# B&R Automation Studio project NAEUL004C00R13L518F00 (part 50)

#### Act_Main.st - Do Not Change!!!
```iecst
(** 2020-05-26 **)
ACTION Act_Main:

	//Main
IF bModuleNotOK = FALSE THEN

		CASE eStat OF

			AWActIdle:
				IF eStatus <> Idle THEN	//Reset Data
					//Private
					fbStop(bEn := FALSE);
					fbRstAxisErr(bEn := FALSE);
					fbJog(bEn := FALSE);
					fbMovRel(bEn := FALSE);
					fbMovAbs(bEn := FALSE);
					fbHoming(bEn := FALSE);
					fbPwrOff(bEn := FALSE);
					fbPwrOn(bEn := FALSE);
					fbFullHm(bEn := FALSE);
					fbFullMovAbs(bEn := FALSE);
					fbFullMovAbsBl(bEn := FALSE);
					fbSDOWrite(bEn := FALSE);
					fbTm(IN := FALSE);
					usiStep				:= 0;
					usiCount			:= 0;
					bNotInterruptible	:= FALSE;
					tyParamOutDriver.uiCtrlword_6040.7	:= FALSE;
					sStatTxt	:= a_sStatText[eStat];

				END_IF

				eStatus	:= Idle;

				IF EDGENEG(p_bManual) THEN
					fMotionCANRstCtrlWord(ADR(tyParamOutDriver));
				END_IF

			AWActGoWidth:
				IF (eStatus = Idle OR eStatus = Busy) THEN

					eStatus	:= Busy;

					sStatTxt	:= a_sStatText[eStat];

					bNotInterruptible	:= TRUE;

					CASE usiStep OF
						0:	//Wait For Motion Parameter Update
							p_diMovePosInUM	:= ABS(fAWWidthToPosInUM(p_diGoWidth , p_diWidthAtHmPos));
							usiStep	:= 1;

						1:	//Check Position Difference
							IF tyParamOut.bPosDiff = TRUE THEN
								usiStep	:= 2;
							ELSE
								eStatus	:= Done;
							END_IF

						2:	//Move
							fbFullMovAbsBl.tyParamInDriver					:= tyParamInDriver;
							fbFullMovAbsBl.tyParamInMove.diPosInUM			:= p_diMovePosInUM;
							fbFullMovAbsBl.tyParamInMove.diDistInUM			:= p_diMoveDistInUM;
							fbFullMovAbsBl.tyParamInMove.diVelInUMPS		:= p_diMoveVelInUMPS;
							fbFullMovAbsBl.tyParamInMove.diAcc				:= p_diMoveAcc;
							fbFullMovAbsBl.tyParamInMove.diDec				:= p_diMoveDec;
							fbFullMovAbsBl.tyParamOut						:= tyParamOut;
							fbFullMovAbsBl(bEn := TRUE);

							IF fbFullMovAbsBl.udiStatus = 0 THEN
								eStatus	:= Done;
							ELSIF fbFullMovAbsBl.udiStatus < 65534 THEN
								eStatus		:= Error;

								IF fbFullMovAbsBl.udiStatus = 1401 THEN
									udiStatus	:= 10002;	//Power On Time Out While Going New Width
								ELSIF fbFullMovAbsBl.udiStatus = 1402 THEN
									udiStatus	:= 10003;	//Homing Time Out While Going New Width
								ELSIF fbFullMovAbsBl.udiStatus = 1403 THEN
									udiStatus	:= 10004;	//Move Absolute Time Out While Going New Width
								ELSIF fbFullMovAbsBl.udiStatus = 1405 THEN
									udiStatus	:= 10005;	//Stop Motion Time Out While Going New Width
								ELSIF fbFullMovAbsBl.udiStatus = 1408 THEN
									udiStatus	:= 10006;	//Axis Error Reset Failed While Going New Width
								ELSIF fbFullMovAbsBl.udiStatus = 1409 THEN
									udiStatus	:= 10007;	//Axis Error Occur In Move Absolute While Going New Width
								ELSIF fbFullMovAbsBl.udiStatus = 1411 THEN
									udiStatus	:= 10008;	//Axis Error Occur In Homing While Going New Width
								ELSIF fbFullMovAbsBl.udiStatus = 1412 THEN
									udiStatus	:= 10009;	//Homing Done But Home Flag Is Not Activated While Going New Width
								ELSIF fbFullMovAbsBl.udiStatus = 1413 THEN
									udiStatus	:= 10010;	//Forward Limit Activated In Homing While Going New Width
								ELSIF fbFullMovAbsBl.udiStatus = 1414 THEN
									udiStatus	:= 10011;	//Reverse Limit Activated In Homing While Going New Width
								ELSIF fbFullMovAbsBl.udiStatus = 1415 THEN
									udiStatus	:= 10012;	//Forward Limit Activated In Move Absolute While Going New Width
								ELSIF fbFullMovAbsBl.udiStatus = 1416 THEN
									udiStatus	:= 10013;	//Reverse Limit Activated In Move Absolute While Going New Width
								ELSE
									udiStatus	:= fbFullMovAbsBl.udiStatus;
								END_IF
							END_IF

					END_CASE

				END_IF

			AWActGoWidthOff:
				IF (eStatus = Idle OR eStatus = Busy) THEN

					eStatus	:= Busy;

					sStatTxt	:= a_sStatText[eStat];

					bNotInterruptible	:= TRUE;

					CASE usiStep OF
						0:	//Wait For Motion Parameter Update
							p_diMovePosInUM	:= ABS(fAWWidthToPosInUM(p_diGoWidth , p_diWidthAtHmPos));
							usiStep	:= 1;

						1:	//Check Position Difference
							IF tyParamOut.bPosDiff = TRUE THEN
								usiStep	:= 2;
							ELSE
								eStatus	:= Done;
							END_IF

						2:	//Move
							fbFullMovAbsBl.tyParamInDriver					:= tyParamInDriver;
							fbFullMovAbsBl.tyParamInMove.diPosInUM			:= p_diMovePosInUM;
							fbFullMovAbsBl.tyParamInMove.diDistInUM			:= p_diMoveDistInUM;
							fbFullMovAbsBl.tyParamInMove.diVelInUMPS		:= p_diMoveVelInUMPS;
							fbFullMovAbsBl.tyParamInMove.diAcc				:= p_diMoveAcc;
							fbFullMovAbsBl.tyParamInMove.diDec				:= p_diMoveDec;
							fbFullMovAbsBl.tyParamOut						:= tyParamOut;
							fbFullMovAbsBl(bEn := TRUE);

							IF fbFullMovAbsBl.udiStatus = 0 THEN
								usiStep	:= 3;
							ELSIF fbFullMovAbsBl.udiStatus < 65534 THEN
								eStatus		:= Error;

								IF fbFullMovAbsBl.udiStatus = 1401 THEN
									udiStatus	:= 10035;	//Power On Time Out While Going New Width And Off
								ELSIF fbFullMovAbsBl.udiStatus = 1402 THEN
									udiStatus	:= 10036;	//Homing Time Out While Going New Width And Off
								ELSIF fbFullMovAbsBl.udiStatus = 1403 THEN
									udiStatus	:= 10037;	//Move Absolute Time Out While Going New Width And Off
								ELSIF fbFullMovAbsBl.udiStatus = 1405 THEN
									udiStatus	:= 10038;	//Stop Motion Time Out While Going New Width And Off
								ELSIF fbFullMovAbsBl.udiStatus = 1408 THEN
									udiStatus	:= 10039;	//Axis Error Reset Failed While Going New Width And Off
								ELSIF fbFullMovAbsBl.udiStatus = 1409 THEN
									udiStatus	:= 10040;	//Axis Error Occur In Move Absolute While Going New Width And Off
								ELSIF fbFullMovAbsBl.udiStatus = 1411 THEN
									udiStatus	:= 10041;	//Axis Error Occur In Homing While Going New Width And Off
								ELSIF fbFullMovAbsBl.udiStatus = 1412 THEN
									udiStatus	:= 10042;	//Homing Done But Home Flag Is Not Activated While Going New Width And Off
								ELSIF fbFullMovAbsBl.udiStatus = 1413 THEN
									udiStatus	:= 10043;	//Forward Limit Activated In Homing While Going New Width And Off
								ELSIF fbFullMovAbsBl.udiStatus = 1414 THEN
									udiStatus	:= 10044;	//Reverse Limit Activated In Homing While Going New Width And Off
								ELSIF fbFullMovAbsBl.udiStatus = 1415 THEN
									udiStatus	:= 10045;	//Forward Limit Activated In Move Absolute While Going New Width And Off
								ELSIF fbFullMovAbsBl.udiStatus = 1416 THEN
									udiStatus	:= 10046;	//Reverse Limit Activated In Move Absolute While Going New Width And Off
								ELSE
									udiStatus	:= fbFullMovAbsBl.udiStatus;
								END_IF
							END_IF

						3:	//Turn Off Motor
							fMotionCANRstCtrlWord(ADR(tyParamOutDriver));
							eStatus	:= Done;

					END_CASE

				END_IF

			AWActFullHm:
				IF (eStatus = Idle OR eStatus = Busy) THEN

					eStatus	:= Busy;

					sStatTxt	:= a_sStatText[eStat];

					bNotInterruptible	:= TRUE;

					fbFullHm.tyParamInDriver	:= tyParamInDriver;
					fbFullHm.tyParamOut			:= tyParamOut;
					fbFullHm(bEn := TRUE);

					IF fbFullHm.udiStatus = 0 THEN
						eStatus	:= Done;
					ELSIF fbFullHm.udiStatus < 65534 THEN
						eStatus		:= Error;

						IF fbFullHm.udiStatus = 1401 THEN
							udiStatus	:= 10014;	//Power On Time Out While Full Homing
						ELSIF fbFullHm.udiStatus = 1402 THEN
							udiStatus	:= 10015;	//Homing Time Out While Full Homing
						ELSIF fbFullHm.udiStatus = 1405 THEN
							udiStatus	:= 10016;	//Stop Motion Time Out While Full Homing
						ELSIF fbFullHm.udiStatus = 1408 THEN
							udiStatus	:= 10017;	//Axis Error Reset Failed While Full Homing
						ELSIF fbFullHm.udiStatus = 1411 THEN
							udiStatus	:= 10018;	//Axis Error Occur In Homing While Full Homing
						ELSIF fbFullHm.udiStatus = 1412 THEN
							udiStatus	:= 10019;	//Homing Done But Home Flag Is Not Activated While Full Homing
						ELSIF fbFullHm.udiStatus = 1413 THEN
							udiStatus	:= 10020;	//Forward Limit Activated In Homing While Full Homing
						ELSIF fbFullHm.udiStatus = 1414 THEN
							udiStatus	:= 10021;	//Reverse Limit Activated In Homing While Full Homing
						ELSE
							udiStatus	:= fbFullHm.udiStatus;
						END_IF
					END_IF

				END_IF

			AWActPwrOn:
				IF (eStatus = Idle OR eStatus = Busy) THEN

					eStatus	:= Busy;

					sStatTxt	:= a_sStatText[eStat];

					fbPwrOn.tyParamInDriver	:= tyParamInDriver;
					fbPwrOn(bEn := TRUE);

					IF fbPwrOn.udiStatus = 0 THEN
						eStatus	:= Done;
					ELSIF fbPwrOn.udiStatus < 65534 THEN
						eStatus		:= Error;

						IF fbPwrOn.udiStatus = 1401 THEN
							udiStatus	:= 10022;	//Power On Time Out
						ELSE
							udiStatus	:= fbPwrOn.udiStatus;
						END_IF
					END_IF

				END_IF

			AWActPwrOff:
				IF (eStatus = Idle OR eStatus = Busy) THEN

					eStatus	:= Busy;

					sStatTxt	:= a_sStatText[eStat];

					fbPwrOff.tyParamInDriver	:= tyParamInDriver;
					fbPwrOff(bEn := TRUE);

					IF fbPwrOff.udiStatus = 0 THEN
						eStatus	:= Done;
					ELSIF fbPwrOff.udiStatus < 65534 THEN
						eStatus		:= Error;

						IF fbPwrOff.udiStatus = 1400 THEN
							udiStatus	:= 10023;	//Power Off Time Out
						ELSE
							udiStatus	:= fbPwrOff.udiStatus;
						END_IF
					END_IF

				END_IF

			AWActHoming:

				IF (eStatus = Idle OR eStatus = Busy) THEN

					eStatus	:= Busy;

					sStatTxt	:= a_sStatText[eStat];

					bNotInterruptible	:= TRUE;

					fbHoming.tyParamInDriver	:= tyParamInDriver;
					fbHoming.tyParamOut			:= tyParamOut;
					fbHoming(bEn := TRUE);

					IF fbHoming.udiStatus = 0 THEN
						eStatus	:= Done;
					ELSIF fbHoming.udiStatus < 65534 THEN
						eStatus		:= Error;

						IF fbHoming.udiStatus = 1402 THEN
							udiStatus	:= 10024;	//Homing Time Out
						ELSIF fbHoming.udiStatus = 1411 THEN
							udiStatus	:= 10018;	//Axis Error Occur In Homing While Full Homing

						ELSIF fbHoming.udiStatus = 1413 THEN
							udiStatus	:= 10020;	//Forward Limit Activated In Homing While Full Homing
						ELSIF fbHoming.udiStatus = 1414 THEN
							udiStatus	:= 10021;	//Reverse Limit Activated In Homing While Full Homing
						ELSE
							udiStatus	:= fbHoming.udiStatus;
						END_IF
					END_IF

				END_IF

			AWActMovAbs:
				IF (eStatus = Idle OR eStatus = Busy) THEN

					eStatus	:= Busy;

					sStatTxt	:= a_sStatText[eStat];

					bNotInterruptible	:= TRUE;

					fbMovAbs.tyParamInDriver			:= tyParamInDriver;
					fbMovAbs.tyParamInMove.diPosInUM	:= p_diMovePosInUM;
					fbMovAbs.tyParamInMove.diDistInUM	:= p_diMoveDistInUM;
					fbMovAbs.tyParamInMove.diVelInUMPS	:= p_diMoveVelInUMPS;
					fbMovAbs.tyParamInMove.diAcc		:= p_diMoveAcc;
					fbMovAbs.tyParamInMove.diDec		:= p_diMoveDec;
					fbMovAbs(bEn := TRUE);

					IF fbMovAbs.udiStatus = 0 THEN
						eStatus	:= Done;
					ELSIF fbMovAbs.udiStatus < 65534 THEN
						eStatus		:= Error;

						IF fbMovAbs.udiStatus = 1403 THEN
							udiStatus	:= 10025;	//Move Absolute Time Out
						ELSE
							udiStatus	:= fbMovAbs.udiStatus;
						END_IF
					END_IF

				END_IF

			AWActMovRel:
				IF (eStatus = Idle OR eStatus = Busy) THEN

					eStatus	:= Busy;

					sStatTxt	:= a_sStatText[eStat];

					bNotInterruptible	:= TRUE;

					fbMovRel.tyParamInDriver			:= tyParamInDriver;
					fbMovRel.tyParamInMove.diPosInUM	:= p_diMovePosInUM;
					fbMovRel.tyParamInMove.diDistInUM	:= p_diMoveDistInUM;
					fbMovRel.tyParamInMove.diVelInUMPS	:= p_diMoveVelInUMPS;
					fbMovRel.tyParamInMove.diAcc		:= p_diMoveAcc;
					fbMovRel.tyParamInMove.diDec		:= p_diMoveDec;
					fbMovRel(bEn := TRUE);

					IF fbMovRel.udiStatus = 0 THEN
						eStatus	:= Done;
					ELSIF fbMovRel.udiStatus < 65534 THEN
						eStatus		:= Error;

						IF fbMovRel.udiStatus = 1404 THEN
							udiStatus	:= 10026;	//Move Relative Time Out
						ELSE
							udiStatus	:= fbMovRel.udiStatus;
						END_IF
					END_IF

				END_IF

			AWActJogOpen:
				IF (eStatus = Idle OR eStatus = Busy) THEN

					eStatus	:= Busy;

					sStatTxt	:= a_sStatText[eStat];

					bNotInterruptible	:= TRUE;

					fbJog.tyParamInDriver	:= tyParamInDriver;
					fbJog.tyParamInMove.diAcc		:= p_diMoveAcc;
					fbJog.tyParamInMove.diDec		:= p_diMoveDec;

					IF p_bDir = TRUE THEN
						fbJog.tyParamInJog.diVelInUMPS	:= p_diJogVelInUMPS * -1;
					ELSE
						fbJog.tyParamInJog.diVelInUMPS	:= p_diJogVelInUMPS;
					END_IF

					fbJog(bEn := TRUE);

					IF fbJog.udiStatus = 0 THEN
						bJogging	:= TRUE;
						bJogOpen	:= TRUE;
						eStatus		:= Done;
					ELSIF fbJog.udiStatus < 65534 THEN
						udiStatus	:= fbJog.udiStatus;
						eStatus		:= Error;
					END_IF

				END_IF

			AWActJogClose:
				IF (eStatus = Idle OR eStatus = Busy) THEN

					eStatus	:= Busy;

					sStatTxt	:= a_sStatText[eStat];

					bNotInterruptible	:= TRUE;

					fbJog.tyParamInDriver			:= tyParamInDriver;
					fbJog.tyParamInMove.diAcc		:= p_diMoveAcc;
					fbJog.tyParamInMove.diDec		:= p_diMoveDec;

					IF p_bDir = TRUE THEN
						fbJog.tyParamInJog.diVelInUMPS	:= p_diJogVelInUMPS;
					ELSE
						fbJog.tyParamInJog.diVelInUMPS	:= p_diJogVelInUMPS * -1;
					END_IF

					fbJog(bEn := TRUE);

					IF fbJog.udiStatus = 0 THEN
						bJogging	:= TRUE;
						bJogClose	:= TRUE;
						eStatus		:= Done;
					ELSIF fbJog.udiStatus < 65534 THEN
						udiStatus	:= fbJog.udiStatus;
						eStatus		:= Error;
					END_IF

				END_IF

			AWActJogStop:
				IF (eStatus = Idle OR eStatus = Busy) THEN

					sStatTxt	:= a_sStatText[eStat];

					fMotionCANJogStop(ADR(tyParamOutDriver));
					bJogging	:= FALSE;
					bJogClose	:= FALSE;
					bJogOpen	:= FALSE;
					eStatus	:= Done;

				END_IF

			AWActRstAxisErr:
				IF (eStatus = Idle OR eStatus = Busy) THEN

					eStatus	:= Busy;

					sStatTxt	:= a_sStatText[eStat];

					fbRstAxisErr(bEn := TRUE);

					IF fbRstAxisErr.udiStatus = 0 THEN
						eStatus	:= Done;
					ELSIF fbRstAxisErr.udiStatus < 65534 THEN
						udiStatus	:= fbRstAxisErr.udiStatus;
						eStatus		:= Error;
					END_IF

				END_IF

			AWActStop:
				IF (eStatus = Idle OR eStatus = Busy) THEN

					eStatus	:= Busy;

					sStatTxt	:= a_sStatText[eStat];

					fbStop.tyParamInDriver	:= tyParamInDriver;
					fbStop(bEn := TRUE);

					IF fbStop.udiStatus = 0 THEN
						bJogging	:= FALSE;
						bJogClose	:= FALSE;
						bJogOpen	:= FALSE;
						eStatus		:= Done;
					ELSIF fbStop.udiStatus < 65534 THEN
						eStatus		:= Error;

						IF fbStop.udiStatus = 1405 THEN
							udiStatus	:= 10027;	//Stop Motion Time Out
						ELSE
							udiStatus	:= fbStop.udiStatus;
						END_IF
					END_IF

				END_IF
		END_CASE
ELSE
	CASE eStat OF
		AWActSDOWrite:
			IF (eStatus = Idle OR eStatus = Busy) THEN

				eStatus	:= Busy;

				sStatTxt	:= a_sStatText[eStat];

				fbTm(IN := TRUE);

				IF fbTm.Q THEN

					fbSDOWrite.tyParamOut	:= tyParamOut;
					fbSDOWrite.tyTuning		:= p_tyTuning;

					fbSDOWrite(bEn := TRUE);

					IF fbSDOWrite.udiStatus = 0 THEN
						eStatus	:= Done;
					ELSIF fbSDOWrite.udiStatus < 65534 THEN
						fMotionCANRstCtrlWord(ADR(tyParamOutDriver));

						IF usiCount < 5 THEN
							fbTm(IN := FALSE);
							fbSDOWrite(bEn := FALSE);

							usiCount	:= usiCount + 1;
						ELSE
							eStatus	:= Error;

							IF fbSDOWrite.udiStatus = 1406 THEN
								udiStatus	:= 10028;	//SDO Write Error
							ELSE
								udiStatus	:= fbSDOWrite.udiStatus;
							END_IF
						END_IF

					END_IF

				END_IF

			END_IF

		AWActBGStartModOKChk:
			IF (eStatus = Idle OR eStatus = Busy) THEN

				sStatTxt	:= a_sStatText[eStat];

				bModuleOKChk	:= TRUE;
				eStatus			:= Done;

			END_IF

		AWActBGStopModOKChk:
			IF (eStatus = Idle OR eStatus = Busy) THEN

				sStatTxt	:= a_sStatText[eStat];

				bModuleOKChk	:= FALSE;
				eStatus			:= Done;

			END_IF

		AWActIdle:
			IF eStatus <> Idle THEN	//Reset Data
				//Private
				fbStop(bEn := FALSE);
				fbRstAxisErr(bEn := FALSE);
				fbJog(bEn := FALSE);
				fbMovRel(bEn := FALSE);
				fbMovAbs(bEn := FALSE);
				fbHoming(bEn := FALSE);
				fbPwrOff(bEn := FALSE);
				fbPwrOn(bEn := FALSE);
				fbFullHm(bEn := FALSE);
				fbFullMovAbs(bEn := FALSE);
				fbFullMovAbsBl(bEn := FALSE);
				fbSDOWrite(bEn := FALSE);
				fbTm(IN := FALSE);
				usiStep				:= 0;
				usiCount			:= 0;
				bNotInterruptible	:= FALSE;
				tyParamOutDriver.uiCtrlword_6040.7	:= FALSE;

				sStatTxt	:= a_sStatText[eStat];

			END_IF

			eStatus	:= Idle;

			IF EDGENEG(p_bManual) THEN
				fMotionCANRstCtrlWord(ADR(tyParamOutDriver));
			END_IF

		AWActRstNode:
			IF (eStatus = Idle OR eStatus = Busy) THEN

				eStatus	:= Busy;

				sStatTxt	:= a_sStatText[eStat];
				IF bRstErr THEN
					fbModuleOK(bEn := FALSE, bModuleOK := bModuleOK);
				END_IF
				fbModuleOK(bEn := TRUE);
				IF fbModuleOK.udiStatus = 0 THEN
					fbModuleOK(bEn := FALSE);
					eStatus			:= Done;
				ELSIF fbModuleOK.udiStatus < 65534 THEN
					eStatus		:= Error;

					IF fbModuleOK.udiStatus = 1407 THEN
						udiStatus	:= 10001;	//CANOpen Communication Error, ModuleOK Not TRUE
						fbModuleOK(bEn := FALSE);
					ELSE
						udiStatus	:= fbModuleOK.udiStatus;
					END_IF
				END_IF
			END_IF

		AWActRstAxisErr:
			IF (eStatus = Idle OR eStatus = Busy) THEN

				eStatus	:= Busy;

				sStatTxt	:= a_sStatText[eStat];

				fbRstAxisErr(bEn := TRUE);

				IF fbRstAxisErr.udiStatus = 0 THEN
					eStatus	:= Done;
				ELSIF fbRstAxisErr.udiStatus < 65534 THEN
					udiStatus	:= fbRstAxisErr.udiStatus;
					eStatus		:= Error;
				END_IF

			END_IF

	END_CASE
END_IF

END_ACTION
```

#### Act_Background.st - Do Not Change!!!
```iecst
(** 2020-05-26 **)
ACTION Act_Background:

	//Update Parameter
	IF bModuleOK = TRUE THEN

		tyParamInMove.diPosInUM		:= p_diMovePosInUM;
		tyParamInMove.diDistInUM	:= p_diMoveDistInUM;
		tyParamInMove.diVelInUMPS	:= p_diMoveVelInUMPS;
		tyParamInMove.diAcc			:= p_diMoveAcc;
		tyParamInMove.diDec			:= p_diMoveDec;

		fMotionCANUpdtDat(ADR(tyParamOut) , p_tyParamInConvert , tyParamOutDriver , tyParamInDriver , tyParamInMove , p_tyParamInHm , p_bDir, p_eNtParamMotorType);

		bWidthPosDiff	:= (tyParamOut.bIsHomed = FALSE) OR ((ABS((ABS(fAWWidthToPosInUM(p_diGoWidth , p_diWidthAtHmPos))) - tyParamOut.diActualPosInUM)) > 500);

		p_tyParamInConvert.diPitchInUM	:= fPitchCalc(p_diWidthOffsetInUM , p_diMaxWidthInUM , p_diMinWidthInUM , p_diPitchInUM);

		fbFullMovAbsBl.tyParamInConvert					:= p_tyParamInConvert;

		IF p_bDir = TRUE THEN
			bOpenSen	:= tyParamOut.bFwdLmtSen;
			bCloseSen	:= tyParamOut.bRevLmtSen;
		ELSE
			bOpenSen	:= tyParamOut.bRevLmtSen;
			bCloseSen	:= tyParamOut.bFwdLmtSen;
		END_IF

		CASE p_eNtParamMotorType OF
			DeltaAsdaA2:
				CASE tyParamOut.udiAxisErrID OF
					8976:	sAxisErrTxt	:= 'Over Current';
					12560:	sAxisErrTxt	:= 'Over Voltage';
					12576:	sAxisErrTxt	:= 'Under Voltage';
					12592:	sAxisErrTxt	:= 'Input Power Phase Loss';
					12816:	sAxisErrTxt	:= 'Regeneration Error';
					12848:	sAxisErrTxt	:= 'Overload';
					12849:	sAxisErrTxt	:= 'Pre-overload Warning';
					13056:	sAxisErrTxt	:= 'U,V,W Wiring Error';
					16912:	sAxisErrTxt	:= 'IGBT Temperature Error';
					21296:	sAxisErrTxt	:= 'Memory Error';
					21569:	sAxisErrTxt	:= 'Emergency Stop Activated';
					21570:	sAxisErrTxt	:= 'Forward Limit Switch Error';
					21571:	sAxisErrTxt	:= 'Reverse Limit Switch Error';
					21572:	sAxisErrTxt	:= 'Forward Software Limit';
					21573:	sAxisErrTxt	:= 'Reverse Software Limit';
					21760:	sAxisErrTxt	:= 'DSP Firmware Upgrade';
					25088:	sAxisErrTxt	:= 'CANopen SYNC Error';
					25360:	sAxisErrTxt	:= 'CANopen Data Initial Error';
					25376:	sAxisErrTxt	:= 'Adjustment Error';
					28961:	sAxisErrTxt	:= 'Motor Protection Error';
					28962:	sAxisErrTxt	:= 'Motor Error';
					29445:	sAxisErrTxt	:= 'Encoder Error';
					29446:	sAxisErrTxt	:= 'Encoder Output Error';
					29968:	sAxisErrTxt	:= 'Serial Communication Error';
					29984:	sAxisErrTxt	:= 'Serial Communication Time Out';
					33024:	sAxisErrTxt	:= 'CANbus Error (Bus-off)';
					33040:	sAxisErrTxt	:= 'CANopen SDO receive buffer overrun';
					33056:	sAxisErrTxt	:= 'CANbus Error (Warning)';
					33072:	sAxisErrTxt	:= 'Node Guarding or Heartbeat Error';
					33280:	sAxisErrTxt	:= 'CANopen PDO Object Error';
					33792:	sAxisErrTxt	:= 'Over Speed';
					34304:	sAxisErrTxt	:= 'Abnormal Pulse Control Command';
					34320:	sAxisErrTxt	:= 'Full Closed Loop Excessive Deviation';
					34321:	sAxisErrTxt	:= 'Excessive Deviation';
				END_CASE

			SchneiderLexium28:
				CASE tyParamOut.udiAxisErrID OF
					8724:	sAxisErrTxt	:= 'Over Current';
					8976:	sAxisErrTxt	:= 'Motor Overload';
					8977:	sAxisErrTxt	:= 'Drive overload (foldback)';
					9088:	sAxisErrTxt	:= 'Calculated offsets for current sensors out OF range';
					9089:	sAxisErrTxt := 'Motor phase missing';
					9090:	sAxisErrTxt := 'Overcurrent detected at one OF the digital outputs';
					12560:	sAxisErrTxt	:= 'DC Bus Over Voltage';
					12576:	sAxisErrTxt	:= 'DC Bus Under Voltage';
					12672:	sAxisErrTxt	:= 'Braking Resistor Overload';
					12673:	sAxisErrTxt	:= 'Safety function Safe Torque Off (STO) triggered';
					12674:	sAxisErrTxt	:= 'DC bus voltage measurement';
					12675:	sAxisErrTxt	:= 'Missing mains supply, undervoltage mains supply';
					12676:	sAxisErrTxt := 'The encoder supply voltage has dropped under operational value';
					12677:	sAxisErrTxt := 'The multi turn encoder battery voltage has dropped under 3 Vdc';
					12678:	sAxisErrTxt := 'Internal position synchronization error	detected between the multi turn AND the single turn modules';
					12679:	sAxisErrTxt := 'Generic error code of the multi turn module is detected';
					12697:	sAxisErrTxt := 'Braking resistor overload';
					16512:	sAxisErrTxt	:= 'Drive overtemperature (IPM)';
					16513:	sAxisErrTxt	:= 'Drive overtemperature (controller)';
					16534:	sAxisErrTxt := 'Temperature sensor inoperative';
					17168:	sAxisErrTxt	:= 'Power stage overtemperature';
					17280:	sAxisErrTxt := 'The encoder temperature is too high';
					17424:	sAxisErrTxt	:= 'Motor overtemperature';
					21808:	sAxisErrTxt	:= 'System error detected (nonvolatilememory)';
					21893:	sAxisErrTxt	:= 'Error detected in non-volatile memory';
					21889:	sAxisErrTxt	:= 'System error detected (nonvolatile memory)';
					21890:	sAxisErrTxt	:= 'System error detected (CAN power supply)';
					21891:	sAxisErrTxt	:= 'System error detected (selftest)';
					21894:	sAxisErrTxt	:= 'System error detected (NV ACCESS)';
					25472:	sAxisErrTxt	:= 'Target position rejected';
					25985:	sAxisErrTxt	:= 'System error detected(FPGA)';
					28816:	sAxisErrTxt	:= 'System error detected (FPGA does NOT match firmware)';
					28817:	sAxisErrTxt	:= 'Emergency Stop Activated';
					28961:	sAxisErrTxt := 'Motor blocked';
					29080:	sAxisErrTxt := 'Commutation error detected';
					29568:  sAxisErrTxt	:= 'Error detected in communication with motor encoder';
					29574:	sAxisErrTxt	:= 'Drive is not synchronous wit master cycle';
					29581:	sAxisErrTxt := 'System error detected (encoder)';
					29587:	sAxisErrTxt	:= 'Encoder overvoltage or overcurrent';
					29592:	sAxisErrTxt := 'The returned position value are no longer considered valid';
					29593:	sAxisErrTxt := 'The multi turn encoder requires an explicit configuration command';
					30081:	sAxisErrTxt := 'Target position rejected';
					30082:	sAxisErrTxt := 'No target values received via the fieldbus';
					33072:	sAxisErrTxt	:= 'CANopen: Heartbeat error detected';
					33296:	sAxisErrTxt := 'R_PDO is too short';
					33921:	sAxisErrTxt	:= 'Actual Motor Velocity Too High';
					33553:	sAxisErrTxt	:= 'Motor torque too high FOR an excessive period OF time';
					33664:	sAxisErrTxt := 'Unstable current loop';
					33922:	sAxisErrTxt := 'Velocity deviation too high';
					34321:	sAxisErrTxt	:= 'Position deviation too high';
					34432:	sAxisErrTxt := 'Position deviation via signal output function MC_OK';
					34441:	sAxisErrTxt := 'Position deviation too high (following error)';
					61568:	sAxisErrTxt	:= 'Fieldbus: Communication	error detected';
					65282:	sAxisErrTxt	:= 'Not possible to read data of electronic motor nameplate';
					65296:	sAxisErrTxt	:= 'Forward Limit Switch Error';
					65297:	sAxisErrTxt	:= 'Reverse Limit Switch Error';
					65281:	sAxisErrTxt := 'System error detected';
					65298:	sAxisErrTxt	:= 'Forward Software Limit';
					65299:	sAxisErrTxt	:= 'Reverse Software Limit';
					65301:	sAxisErrTxt := 'The encoder firmware cannot operate on the provided hardware';

				END_CASE

			EstunPronet:
				CASE tyParamOut.udiAxisErrID OF
					65281:	sAxisErrTxt	:= 'Parameter breakdown';//A01
					65282:	sAxisErrTxt	:= 'AD shift channels breakdown';
					65283:	sAxisErrTxt	:= 'Overspeed';
					65284:	sAxisErrTxt	:= 'Overload';
					65285:	sAxisErrTxt := 'Position error counteroverflow ';
					65286:	sAxisErrTxt := 'Position error pulse overflow';
					65287:	sAxisErrTxt	:= 'The setting of electronic gear or given pulse frequency is not reasonable';
					65288:	sAxisErrTxt	:= 'The 1st channel of current detection is wrong.';
					65289:	sAxisErrTxt	:= 'The 2nd channel of current detection is wrong.';
					65290:	sAxisErrTxt	:= 'Incremental Encoder is break off.';//A10
					65292:	sAxisErrTxt	:= 'Overcurrent';
					65293:	sAxisErrTxt	:= 'Overvoltage';
					65294:	sAxisErrTxt	:= 'Undervoltage';
					65295:	sAxisErrTxt := 'Bleeder resistor error';
					65296:	sAxisErrTxt := 'Regeneration error';
					65297:	sAxisErrTxt := 'Resolver error';
					65298:	sAxisErrTxt := 'IGBT superheat alarm';
					65299:	sAxisErrTxt := 'Motor overheat alarm';
					65300:	sAxisErrTxt := 'Power line phase shortage';//A20
					65301:	sAxisErrTxt	:= 'Instantaneous power off alarm';
					65302:	sAxisErrTxt	:= 'Motor temperature detection sensor is break off.';
					65303:	sAxisErrTxt := 'Brake overcurrent alarm';//A23
					65305:	sAxisErrTxt := 'Motor power line U overcurrent';//A25
					65306:	sAxisErrTxt := 'Motor power line V overcurrent';//A26
					65307:	sAxisErrTxt := 'Motor power line W overcurrent';//A27
					65322:	sAxisErrTxt	:= 'Servomotor type error';//A42
					65323:	sAxisErrTxt	:= 'Servo drive type error';
					65325:	sAxisErrTxt	:= 'Absolute encoder multiturn information error';
					65326:	sAxisErrTxt	:= 'Absolute encoder multiturn information overflow';
					65327:	sAxisErrTxt	:= 'Battery voltage below 2.5V';
					65328:	sAxisErrTxt	:= 'Battery voltage below 3.1V';//A48
					65330:	sAxisErrTxt := 'Serial encoder communication overtime ';//A50
					65331:	sAxisErrTxt := 'Absolute encoder overspeed alarm detected';
					65332:  sAxisErrTxt	:= 'Absolute state of serial encoder error';
					65333:	sAxisErrTxt	:= 'Serial encoder calcaution error';
					65334:	sAxisErrTxt := 'Parity bit or end bit in serial encoder control domain error';
					65335:	sAxisErrTxt	:= 'Serial encoder communication data checking error';
					65336:	sAxisErrTxt := 'End bit in serial encoder control domain error';
					65338:	sAxisErrTxt := 'Serial encoder data empty';
					65339:	sAxisErrTxt := 'Serial encoder data format error';
					65340:	sAxisErrTxt := 'Communication module not detected ';//A60
					65341:	sAxisErrTxt := 'Communication unsuccessful';
					65342:	sAxisErrTxt := 'Servo drive can not receive the period data of communication module ';
					65343:	sAxisErrTxt := 'Communication module can not receive the servo drive response data.';
					65344:	sAxisErrTxt := 'Communication module and bus connectionless';
					65346:	sAxisErrTxt := 'CAN communication abnormal';
					65347:	sAxisErrTxt := 'Receiving heartbeat timeout';
					65349:	sAxisErrTxt := 'Synchronization signal monitoring cycle is longer than setting';
					65362: sAxisErrTxt	:= 'Torque output alarm';
				END_CASE
		END_CASE

	ELSE

		tyParamOut.bAxisErr			:= FALSE;
		tyParamOut.bFwdLmtSen		:= FALSE;
		tyParamOut.bInPos			:= FALSE;
		tyParamOut.bIsHomed			:= FALSE;
		tyParamOut.bPosDiff			:= TRUE;
		tyParamOut.bPwrOn			:= FALSE;
		tyParamOut.bRevLmtSen		:= FALSE;
		tyParamOut.bStopped			:= TRUE;
		tyParamOut.diActualPosInUM	:= 0;
		tyParamOut.diHmAcc			:= 0;
		tyParamOut.diHmSpdForSwitch	:= 0;
		tyParamOut.diHmSpdForZero	:= 0;
		tyParamOut.diProfileAcc		:= 0;
		tyParamOut.diProfileDec		:= 0;
		tyParamOut.udiAxisErrID		:= 0;

		bWidthPosDiff				:= TRUE;

	END_IF

	//Abnormal Movement
	IF eStatus1 <> Error THEN
		IF p_bOps = TRUE AND eStatus = Idle THEN
			IF (ABS(tyParamOut.diActualPosInUM - diActualPosInUMOld) > 2000) AND (ABS(tyParamOut.diActualPosInUM - diActualPosInUMOld) < 10000) THEN
				eStatus1	:= Error;
				udiStatus1	:= 10000;	//Axis Move Abnormally By External Force

				fMotionCANRstCtrlWord(ADR(tyParamOutDriver));
				p_eAct	:= AWActIdle;
				eStat	:= AWActIdle;
			END_IF
		ELSE
			diActualPosInUMOld	:= tyParamOut.diActualPosInUM;
		END_IF
	END_IF

	//Reset Error
	IF (eStatus1 = Error) AND bRstErr THEN
		eStatus1	:= Idle;
		udiStatus1	:= 0;
	END_IF

	//Request Position To Movement Out Of Range
	IF p_bOps
		AND((tyParamInMove.diPosInUM < p_diMinAbsPosInUM) OR (tyParamInMove.diPosInUM > p_diMaxAbsPosInUM))
		AND (eStatus2 <> Error) THEN
		eStatus2	:= Error;
		udiStatus2	:= 10029;	//Request Absolute Position Out Of Range

		fMotionCANRstCtrlWord(ADR(tyParamOutDriver));
		p_eAct	:= AWActIdle;
		eStat	:= AWActIdle;
	END_IF

	//Reset Error
	IF (eStatus2 = Error) AND bRstErr THEN
		eStatus2	:= Idle;
		udiStatus2	:= 0;
	END_IF

	//Sensor Interrupt
	IF (bNotInterruptible = TRUE OR bJogging) AND eStatus3 <> Error THEN

		IF p_bInletSensor = TRUE THEN
			eStatus3	:= Error;
			udiStatus3	:= 10030;	//Inlet Sensor Interrupt Auto Width Movement

			fMotionCANRstCtrlWord(ADR(tyParamOutDriver));
			p_eAct	:= AWActIdle;
			eStat	:= AWActIdle;

		ELSIF p_bOutletSensor = TRUE THEN
			eStatus3	:= Error;
			udiStatus3	:= 10031;	//Outlet Sensor Interrupt Auto Width Movement

			fMotionCANRstCtrlWord(ADR(tyParamOutDriver));
			p_eAct	:= AWActIdle;
			eStat	:= AWActIdle;

		ELSIF p_bClearSensor = TRUE THEN
			eStatus3	:= Error;
			udiStatus3	:= 10032;	//Clear Sensor Interrupt Auto Width Movement

			fMotionCANRstCtrlWord(ADR(tyParamOutDriver));
			p_eAct	:= AWActIdle;
			eStat	:= AWActIdle;

		ELSIF p_bMiddleSensor = TRUE THEN
			eStatus3	:= Error;
			udiStatus3	:= 10033;	//Middle Sensor Interrupt Auto Width Movement

			fMotionCANRstCtrlWord(ADR(tyParamOutDriver));
			p_eAct	:= AWActIdle;
			eStat	:= AWActIdle;

		ELSIF p_bInterruptSensor = TRUE THEN
			eStatus3	:= Error;
			udiStatus3	:= 10034;	//Sensor Interrupt Auto Width Movement

			fMotionCANRstCtrlWord(ADR(tyParamOutDriver));
			p_eAct	:= AWActIdle;
			eStat	:= AWActIdle;

		ELSIF p_bCloseInterruptSensor = TRUE AND bJogOpen = FALSE THEN
			eStatus3	:= Error;
			udiStatus3	:= 10047;	//Sensor Interrupt Auto Width Movement

			fMotionCANRstCtrlWord(ADR(tyParamOutDriver));
			p_eAct	:= AWActIdle;
			eStat	:= AWActIdle;

		ELSIF p_bOpenInterruptSensor = TRUE AND bJogClose = FALSE THEN
			eStatus3	:= Error;
			udiStatus3	:= 10048;	//Sensor Interrupt Auto Width Movement

			fMotionCANRstCtrlWord(ADR(tyParamOutDriver));
			p_eAct	:= AWActIdle;
			eStat	:= AWActIdle;
		END_IF

	END_IF

	//Reset Error
	IF (eStatus3 = Error AND bRstErr)
		OR (p_bOpenInterruptSensor AND eStat = AWActJogClose)
		OR (p_bCloseInterruptSensor AND eStat = AWActJogOpen)
		THEN
		eStatus3	:= Idle;
		udiStatus3	:= 0;
	END_IF

	IF bRstErr THEN
		udiStatus	:= 0;
		bJogging	:= FALSE;
		bJogClose	:= FALSE;
		bJogOpen	:= FALSE;
	END_IF

	fbServoModuleOk(IN:= bModuleOK);
	fbServoModuleNotOk(IN:= bModuleOK = FALSE);
	IF fbServoModuleNotOk.Q AND udiStatus <> 10001 THEN

		bModuleNotOK		:= TRUE;
		bModuleNotOKLock	:= TRUE;
		usiRstStep	:= 0;
		tyParamOutDriver.uiCtrlword_6040	:= 0;
		tyParamOutDriver.siModOfOpt_6060	:= 0;
		tyParamOutDriver.diTargetPos_607A	:= 0;
		tyParamOutDriver.udiMoveSpd_6081	:= 0;
		tyParamOutDriver.siHmMethod_6098	:= 0;
		tyParamOutDriver.diJogVel_60FF		:= 0;

		CASE p_eNtParamMotorType OF

			DeltaAsdaA2:
				fbModuleOK(bModuleOK:= FALSE);
				IF eStatus = Idle THEN
					eAct	:= AWActRstNode;
				END_IF

				IF (eStatus = Done OR eStatus = Error)AND eStat = AWActRstNode THEN

					eAct	:= AWActIdle;
				END_IF

			EstunPronet:
				fbModuleOK(bModuleOK:= FALSE);
				IF eStatus = Idle THEN
					eAct	:= AWActRstNode;
				END_IF

				IF (eStatus = Done OR eStatus = Error)AND eStat = AWActRstNode THEN

					eAct	:= AWActIdle;
				END_IF

			SchneiderLexium28:
			// Do Nothing
		END_CASE

	ELSIF bModuleNotOK = TRUE AND fbServoModuleOk.Q THEN

		CASE usiRstStep OF

			0:
				IF eStatus = Idle THEN
					eAct	:= AWActRstAxisErr;
				END_IF

				IF eStatus = Done AND eStat = AWActRstAxisErr THEN
					eAct	:= AWActIdle;
					usiRstStep	:= 4;
				END_IF

			4: tyParamOutDriver.siModOfOpt_6060 := 1;
				usiRstStep	:= 5;

			5: tyParamOutDriver.siModOfOpt_6060 := 1;
				fbRstNodeTimer(IN:=TRUE);

				IF tyParamInDriver.siModOfOptDisp_6061 = 1 THEN
					usiRstStep	:= 6;
					fbRstNodeTimer(IN:=FALSE);
				ELSIF fbRstNodeTimer.Q THEN
					usiRstStep	:= 8;
					fbRstNodeTimer(IN:=FALSE);
				END_IF

			6: tyParamOutDriver.siModOfOpt_6060 := 6;
				fbRstNodeTimer(IN:=FALSE);
				usiRstStep	:= 7;

			7: tyParamOutDriver.siModOfOpt_6060 := 6;
				fbRstNodeTimer(IN:=TRUE);

				IF tyParamInDriver.siModOfOptDisp_6061 = 6 THEN
					usiRstStep	:= 10;
					fbRstNodeTimer(IN:=FALSE);
				ELSIF fbRstNodeTimer.Q THEN
					usiRstStep	:= 9;
					fbRstNodeTimer(IN:=FALSE);
				END_IF

			8:	fbModuleOK(bEn := TRUE, bModuleOK:= FALSE);
				fbRstNodeTimer(IN:=FALSE);
				usiRstStep	:= 9;

			9:	fbModuleOK(bModuleOK:= FALSE);
				IF eStatus = Idle THEN
					eAct	:=AWActRstNode;
				END_IF

				IF eStatus = Done AND eStat = AWActRstNode THEN
					usiRstStep	:= 0;
					eAct		:= AWActIdle;
				END_IF

			10:IF eStatus = Idle THEN
					eAct	:= AWActRstAxisErr;
				END_IF

				IF eStatus = Done AND eStat = AWActRstAxisErr THEN
					eAct			:=AWActIdle;
					usiRstStep	:= 11;
				END_IF

			11:

				IF eStatus = Idle THEN
					eAct	:= AWActSDOWrite;
				END_IF

				IF eStatus = Done AND eStat = AWActSDOWrite THEN
					eAct			:= AWActIdle;
					usiRstStep	:= 13;

				ELSIF udiStatus = 10028 THEN
					eAct			:= AWActIdle;
					usiRstStep	:= 0;
				END_IF

			13: bModuleNotOK	:= FALSE;
				usiRstStep	:= 0;
		END_CASE
	ELSE
		eAct	:= AWActIdle;

	END_IF

	IF tyParamOut.bPosDiff = FALSE THEN
		tyParamOutDriver.uiCtrlword_6040.4	:= FALSE;
	END_IF

END_ACTION
```

#### Act_Alarm.st - Do Not Change!!!
```iecst
(** 2020-03-16 **)
ACTION Act_Alarm:

	//Error
	IF EDGEPOS(eStatus = Error) THEN

		tyAlmData.sProgNm		:= p_sProgNm;
		tyAlmData.udiCode		:= udiStatus;
		tyAlmData.eSeverity		:= AlmSeverityError;
		tyAlmData.udiRunTime	:= tyAlmData.udiRunTime + 1;
		tyAlmData.bAlm			:= TRUE;
		tyAlmData.udiModuleNum  := udiModuleNum;
		g_sAWOpenProgNm			:= p_sProgNm;
		//Get Error Message
		IF tyAlmData.udiCode < 10000 OR tyAlmData.udiCode > 10299 THEN
			tyAlmData.sAlmMsg	:= 'Unknown';
			tyAlmData.sRcyMsg	:= 'Unknown';
		ELSE
			tyAlmData.sAlmMsg	:= a_tyAlmText[tyAlmData.udiCode].sAlmText;
			tyAlmData.sRcyMsg	:= a_tyAlmText[tyAlmData.udiCode].sRcyText;
		END_IF

		sStatTxt	:= tyAlmData.sAlmMsg;

	ELSIF bRstErr AND (tyAlmData.udiCode <> 0) THEN

		tyAlmData.udiCode	:= 0;
		tyAlmData.eSeverity	:= AlmSeverityNA;
		tyAlmData.sAlmMsg	:= '';
		tyAlmData.sRcyMsg	:= '';
		tyAlmData.bAlm			:= FALSE;
		sStatTxt	:= a_sStatText[eStat];

	END_IF

END_ACTION
```

#### Act_Alarm1.st - Do Not Change!!!
```iecst
(** 2020-03-16 **)
ACTION Act_Alarm1:

	//Error
	IF EDGEPOS(eStatus1 = Error) THEN

		tyAlmData1.sProgNm		:= p_sProgNm;
		tyAlmData1.udiCode		:= udiStatus1;
		tyAlmData1.eSeverity	:= AlmSeverityError;
		tyAlmData1.udiRunTime	:= tyAlmData1.udiRunTime + 1;
		tyAlmData1.bAlm			:= TRUE;
		tyAlmData1.udiModuleNum  := udiModuleNum;
		g_sAWOpenProgNm			:= p_sProgNm;
		//Get Error Message
		IF tyAlmData1.udiCode < 10000 OR tyAlmData1.udiCode > 10099 THEN
			tyAlmData1.sAlmMsg	:= 'Unknown';
			tyAlmData1.sRcyMsg	:= 'Unknown';
		ELSE
			tyAlmData1.sAlmMsg	:= a_tyAlmText[tyAlmData1.udiCode].sAlmText;
			tyAlmData1.sRcyMsg	:= a_tyAlmText[tyAlmData1.udiCode].sRcyText;
		END_IF

		sStatTxt	:= tyAlmData1.sAlmMsg;

	ELSIF bRstErr AND (tyAlmData1.udiCode <> 0) THEN

		tyAlmData1.udiCode		:= 0;
		tyAlmData1.eSeverity	:= AlmSeverityNA;
		tyAlmData1.sAlmMsg		:= '';
		tyAlmData1.sRcyMsg		:= '';
		tyAlmData1.bAlm			:= FALSE;
		sStatTxt	:= a_sStatText[eStat];

	END_IF

END_ACTION
```

#### Act_Alarm2.st - Do Not Change!!!
```iecst
(** 2020-03-16 **)
ACTION Act_Alarm2:

	//Error
	IF EDGEPOS(eStatus2 = Error) THEN

		tyAlmData2.sProgNm		:= p_sProgNm;
		tyAlmData2.udiCode		:= udiStatus2;
		tyAlmData2.eSeverity	:= AlmSeverityError;
		tyAlmData2.udiRunTime	:= tyAlmData2.udiRunTime + 1;
		tyAlmData2.bAlm			:= TRUE;
		tyAlmData2.udiModuleNum  := udiModuleNum;
		g_sAWOpenProgNm			:= p_sProgNm;
		//Get Error Message
		IF tyAlmData2.udiCode < 10000 OR tyAlmData2.udiCode > 10099 THEN
			tyAlmData2.sAlmMsg	:= 'Unknown';
			tyAlmData2.sRcyMsg	:= 'Unknown';
		ELSE
			tyAlmData2.sAlmMsg	:= a_tyAlmText[tyAlmData2.udiCode].sAlmText;
			tyAlmData2.sRcyMsg	:= a_tyAlmText[tyAlmData2.udiCode].sRcyText;
		END_IF

		sStatTxt	:= tyAlmData2.sAlmMsg;

	ELSIF bRstErr AND (tyAlmData2.udiCode <> 0) THEN

		tyAlmData2.udiCode		:= 0;
		tyAlmData2.eSeverity	:= AlmSeverityNA;
		tyAlmData2.sAlmMsg		:= '';
		tyAlmData2.sRcyMsg		:= '';
		tyAlmData2.bAlm			:= FALSE;
		sStatTxt	:= a_sStatText[eStat];

	END_IF

END_ACTION
```

#### Act_Alarm3.st - Do Not Change!!!
```iecst
(** 2020-03-16 **)
ACTION Act_Alarm3:

	//Error
	IF EDGEPOS(eStatus3 = Error) THEN

		tyAlmData3.sProgNm		:= p_sProgNm;
		tyAlmData3.udiCode		:= udiStatus3;
		tyAlmData3.eSeverity	:= AlmSeverityError;
		tyAlmData3.udiRunTime	:= tyAlmData3.udiRunTime + 1;
		tyAlmData3.bAlm			:= TRUE;
		tyAlmData3.udiModuleNum  := udiModuleNum;
		g_sAWOpenProgNm			:= p_sProgNm;
		//Get Error Message
		IF tyAlmData3.udiCode < 10000 OR tyAlmData3.udiCode > 10099 THEN
			tyAlmData3.sAlmMsg	:= 'Unknown';
			tyAlmData3.sRcyMsg	:= 'Unknown';
		ELSE
			tyAlmData3.sAlmMsg	:= a_tyAlmText[tyAlmData3.udiCode].sAlmText;
			tyAlmData3.sRcyMsg	:= a_tyAlmText[tyAlmData3.udiCode].sRcyText;
		END_IF

		sStatTxt	:= tyAlmData3.sAlmMsg;

	ELSIF bRstErr AND (tyAlmData3.udiCode <> 0) THEN

		tyAlmData3.udiCode		:= 0;
		tyAlmData3.eSeverity	:= AlmSeverityNA;
		tyAlmData3.sAlmMsg		:= '';
		tyAlmData3.sRcyMsg		:= '';
		tyAlmData3.bAlm			:= FALSE;
		sStatTxt	:= a_sStatText[eStat];

	END_IF

END_ACTION
```

#### InputRef.var - Do Not Change!!!
```iecst
(*2020-05-26*)
(**)
(*General*)
VAR
	p_eAct : REFERENCE TO eAWAction;
	p_udiRstErr : REFERENCE TO UDINT;
	p_bPrep : REFERENCE TO BOOL;
	p_bEn : REFERENCE TO BOOL;
	p_bDis : REFERENCE TO BOOL;
END_VAR
(**)
(*Configuration*)
VAR
	p_bOps : REFERENCE TO BOOL;
	p_bManual : REFERENCE TO BOOL;
	p_diWidthAtHmPos : REFERENCE TO DINT;
	p_tyTuning : REFERENCE TO tyMotionCANTuning;
	p_diGoWidth : REFERENCE TO DINT;
	p_diJogVelInUMPS : REFERENCE TO DINT;
	p_diMovePosInUM : REFERENCE TO DINT;
	p_diMoveDistInUM : REFERENCE TO DINT;
	p_diMoveVelInUMPS : REFERENCE TO DINT;
	p_diMoveAcc : REFERENCE TO DINT;
	p_diMoveDec : REFERENCE TO DINT;
	p_diMinAbsPosInUM : REFERENCE TO DINT;
	p_diMaxAbsPosInUM : REFERENCE TO DINT;
	p_diMinWidthInUM : REFERENCE TO DINT;
	p_diMaxWidthInUM : REFERENCE TO DINT;
	p_diWidthOffsetInUM : REFERENCE TO DINT;
	p_bInletSensor : REFERENCE TO BOOL;
	p_bOutletSensor : REFERENCE TO BOOL;
	p_bClearSensor : REFERENCE TO BOOL;
	p_bMiddleSensor : REFERENCE TO BOOL;
	p_bInterruptSensor : REFERENCE TO BOOL;
	p_bOpenInterruptSensor : REFERENCE TO BOOL;
	p_bCloseInterruptSensor : REFERENCE TO BOOL;
	p_bSafetyInterruptSen : REFERENCE TO BOOL;
	p_bDir : REFERENCE TO BOOL;
	p_bDirBl : REFERENCE TO BOOL;
	p_bNoIndexPulse : REFERENCE TO BOOL;
	p_usiNode : REFERENCE TO USINT;
	p_sDevice : REFERENCE TO STRING[3];
	p_sProgNm : REFERENCE TO STRING[15];
	p_diMoveBacklashDistInUM : REFERENCE TO DINT;
	p_diPitchInUM : REFERENCE TO DINT;
	p_tyParamInHm : REFERENCE TO tyMotionCANParamInHm;
	p_tyParamInConvert : REFERENCE TO tyMotionCANParamInConvert;
	p_bNtSettingsLoadDone : REFERENCE TO BOOL;
	p_eNtParamMotorType : REFERENCE TO eServoMotorType;
	p_bOutletShutterCloseRS : REFERENCE TO BOOL;
	p_bOutletShutterCloseRS2 : REFERENCE TO BOOL;
	p_bOutletShutterCloseRS3 : REFERENCE TO BOOL;
	p_bProjInletShutPrep : REFERENCE TO BOOL;
	p_bInShutterDis : REFERENCE TO BOOL;
	p_bOutShutterDis : REFERENCE TO BOOL;
	p_bProjOutletShutPrep : REFERENCE TO BOOL;
	p_bInletShutterCloseRS : REFERENCE TO BOOL;
	p_bUITeachServo : REFERENCE TO BOOL;
	p_bPusherRetSen : REFERENCE TO BOOL;
	p_bPusherExtSen : REFERENCE TO BOOL;
END_VAR
```

#### Local.var - Do Not Change!!!
```iecst
(*2020-05-26*)
(**)
(*Local Action, State & Status*)
VAR
	eAct : eAWAction := AWActIdle;
	eStat : eAWAction := AWActIdle;
	eMainStatus : eFBStatus := Idle;
	eStatus : eFBStatus := Idle;
	eStatus1 : eFBStatus := Idle;
	eStatus2 : eFBStatus := Idle;
	eStatus3 : eFBStatus := Idle;
	udiStatus : UDINT := 0;
	udiStatus1 : UDINT := 0;
	udiStatus2 : UDINT := 0;
	udiStatus3 : UDINT := 0;
	sStatTxt : STRING[200] := '';
	a_sStatText : ARRAY[0..50] OF STRING[200] := ['Idling','Going Width','Full Homing','Powering On','Powering Off','Homing','Moving Absolute','Moving Relative','Jogging Open','Jogging Close','Jogging Stop','Resetting Axis Error','Stopping','Writing SDO','Background Starting Module OK Check','Background Stopping Module OK Check','Going Width And Power Off','Reset Servo Module Node',33('')];
END_VAR
(**)
(*Local Alarm*)
VAR
	tyAlmData : tyAlmDat;
	tyAlmData1 : tyAlmDat;
	tyAlmData2 : tyAlmDat;
	tyAlmData3 : tyAlmDat;
	a_tyAlmText : ARRAY[10000..10299] OF tyAlmTxt := [(sAlmText:='Axis Move Abnormally By External Force',sRcyText:='Servo Motor Abnormal Operation. Reset And Resume Operation. If The Problem Persists, Please Contact Nutek For A Possible Solution.'),(sAlmText:='CANOpen Communication Error, ModuleOK Not TRUE',sRcyText:='Fail While Read/Write Data. Reset The Error And Resume Operation.'),(sAlmText:='Power On Time Out While Going New Width',sRcyText:='Timeout Expired Before Operation Completed. Reset And Resume Operation.'),(sAlmText:='Homing Time Out While Going New Width',sRcyText:='Timeout Expired Before Operation Completed. Reset And Resume Operation.'),(sAlmText:='Move Absolute Time Out While Going New Width',sRcyText:='Timeout Expired Before Operation Completed. Reset And Resume Operation.'),(sAlmText:='Stop Motion Time Out While Going New Width',sRcyText:='Timeout Expired Before Operation Completed. Reset And Resume Operation.'),(sAlmText:='Axis Error Reset Failed While Going New Width',sRcyText:='Axis Error Reset Failed. Please Retry Again Reset Operation. If The Problem Persists, Please Contact Nutek For A Possible Solution.'),(sAlmText:='Axis Error Occur In Move Absolute While Going New Width',sRcyText:='Servo Motor Abnormal Operation. Reset And Resume Operation. If The Problem Persists, Please Contact Nutek For A Possible Solution.'),(sAlmText:='Axis Error Occur In Homing While Going New Width',sRcyText:='Servo Motor Abnormal Operation. Reset And Resume Operation. If The Problem Persists, Please Contact Nutek For A Possible Solution.'),(sAlmText:='Homing Done But Home Flag Is Not Activated While Going New Width',sRcyText:='Servo Motor Abnormal Operation. Reset And Resume Operation. If The Problem Persists, Please Contact Nutek For A Possible Solution.'),(sAlmText:='Forward Limit Activated In Homing While Going New Width',sRcyText:='Forward Limit Switch Is Activated. Reset The Error By Operate The Motor Backwards.'),(sAlmText:='Reverse Limit Activated In Homing While Going New Width',sRcyText:='Reverse Limit Switch Is Activated. Reset The Error By Operate The Motor Backwards.'),(sAlmText:='Forward Limit Activated In Move Absolute While Going New Width',sRcyText:='Forward Limit Switch Is Activated. Reset The Error By Operate The Motor Backwards.'),(sAlmText:='Reverse Limit Activated In Move Absolute While Going New Width',sRcyText:='Reverse Limit Switch Is Activated. Reset The Error By Operate The Motor Backwards.'),(sAlmText:='Power On Time Out While Full Homing',sRcyText:='Timeout Expired Before Operation Completed. Reset And Resume Operation.'),(sAlmText:='Homing Time Out While Full Homing',sRcyText:='Timeout Expired Before Operation Completed. Reset And Resume Operation.'),(sAlmText:='Stop Motion Time Out While Full Homing',sRcyText:='Timeout Expired Before Operation Completed. Reset And Resume Operation.'),(sAlmText:='Axis Error Reset Failed While Full Homing',sRcyText:='Axis Error Reset Failed. Please Retry Again Reset Operation. If The Problem Persists, Please Contact Nutek For A Possible Solution.'),(sAlmText:='Axis Error Occur In Homing While Full Homing',sRcyText:='Servo Motor Abnormal Operation. Reset And Resume Operation. If The Problem Persists, Please Contact Nutek For A Possible Solution.'),(sAlmText:='Homing Done But Home Flag Is Not Activated While Full Homing',sRcyText:='Servo Motor Abnormal Operation. Reset And Resume Operation. If The Problem Persists, Please Contact Nutek For A Possible Solution.'),(sAlmText:='Forward Limit Activated In Homing While Full Homing',sRcyText:='Forward Limit Switch Is Activated. Reset The Error By Operate The Motor Backwards.'),(sAlmText:='Reverse Limit Activated In Homing While Full Homing',sRcyText:='Reverse Limit Switch Is Activated. Reset The Error By Operate The Motor Backwards.'),(sAlmText:='Power On Time Out',sRcyText:='Timeout Expired Before Operation Completed. Reset And Resume Operation.'),(sAlmText:='Power Off Time Out',sRcyText:='Timeout Expired Before Operation Completed. Reset And Resume Operation.'),(sAlmText:='Homing Time Out',sRcyText:='Timeout Expired Before Operation Completed. Reset And Resume Operation.'),(sAlmText:='Move Absolute Time Out',sRcyText:='Timeout Expired Before Operation Completed. Reset And Resume Operation.'),(sAlmText:='Move Relative Time Out',sRcyText:='Timeout Expired Before Operation Completed. Reset And Resume Operation.'),(sAlmText:='Stop Motion Time Out',sRcyText:='Timeout Expired Before Operation Completed. Reset And Resume Operation.'),(sAlmText:='SDO Write Error',sRcyText:='Fail While Write Data. Reset The Error And Resume Operation.'),(sAlmText:='Request Absolute Position Out Of Range',sRcyText:='Request Absolute Position Does Not Fall Within The Expected Range.'),(sAlmText:='Inlet Sensor Interrupt Auto Width Movement',sRcyText:='Operation Stop Due To The Interruption Of Sensor While Auto Width Moving. Solve The Interruption To Resume Operation.'),(sAlmText:='Outlet Sensor Interrupt Auto Width Movement',sRcyText:='Operation Stop Due To The Interruption Of Sensor While Auto Width Moving. Solve The Interruption To Resume Operation.'),(sAlmText:='Clear Sensor Interrupt Auto Width Movement',sRcyText:='Operation Stop Due To The Interruption Of Sensor While Auto Width Moving. Solve The Interruption To Resume Operation.'),(sAlmText:='Middle Sensor Interrupt Auto Width Movement',sRcyText:='Operation Stop Due To The Interruption Of Sensor While Auto Width Moving. Solve The Interruption To Resume Operation.'),(sAlmText:='Sensor Interrupt Auto Width Movement',sRcyText:='Operation Stop Due To The Interruption Of Sensor While Auto Width Moving. Solve The Interruption To Resume Operation.'),(sAlmText:='Power On Time Out While Going New Width And Off',sRcyText:='Timeout Expired Before Operation Completed. Reset And Resume Operation.'),(sAlmText:='Homing Time Out While Going New Width And Off',sRcyText:='Timeout Expired Before Operation Completed. Reset And Resume Operation.'),(sAlmText:='Move Absolute Time Out While Going New Width And Off',sRcyText:='Timeout Expired Before Operation Completed. Reset And Resume Operation.'),(sAlmText:='Stop Motion Time Out While Going New Width And Off',sRcyText:='Timeout Expired Before Operation Completed. Reset And Resume Operation.'),(sAlmText:='Axis Error Reset Failed While Going New Width And Off',sRcyText:='Axis Error Reset Failed. Please Retry Again Reset Operation. If The Problem Persists, Please Contact Nutek For A Possible Solution.'),(sAlmText:='Axis Error Occur In Move Absolute While Going New Width And Off',sRcyText:='Servo Motor Abnormal Operation. Reset And Resume Operation. If The Problem Persists, Please Contact Nutek For A Possible Solution.'),(sAlmText:='Axis Error Occur In Homing While Going New Width And Off',sRcyText:='Servo Motor Abnormal Operation. Reset And Resume Operation. If The Problem Persists, Please Contact Nutek For A Possible Solution.'),(sAlmText:='Homing Done But Home Flag Is Not Activated While Going New Width And Off',sRcyText:='Servo Motor Abnormal Operation. Reset And Resume Operation. If The Problem Persists, Please Contact Nutek For A Possible Solution.'),(sAlmText:='Forward Limit Activated In Homing While Going New Width And Off',sRcyText:='Forward Limit Switch Is Activated. Reset The Error By Operate The Motor Backwards.'),(sAlmText:='Reverse Limit Activated In Homing While Going New Width And Off',sRcyText:='Reverse Limit Switch Is Activated. Reset The Error By Operate The Motor Backwards.'),(sAlmText:='Forward Limit Activated In Move Absolute While Going New Width And Off',sRcyText:='Forward Limit Switch Is Activated. Reset The Error By Operate The Motor Backwards.'),(sAlmText:='Reverse Limit Activated In Move Absolute While Going New Width And Off',sRcyText:='Reverse Limit Switch Is Activated. Reset The Error By Operate The Motor Backwards.'),2((sAlmText:='Sensor Interrupt Auto Width Movement',sRcyText:='Operation Stop Due To The Interruption Of Sensor While Auto Width Moving. Solve The Interruption To Resume Operation.')),249((0)),(sAlmText:='Forward Limit Activated',sRcyText:='Forward Limit Switch Is Activated. Reset The Error By Operate The Motor Backwards.'),(sAlmText:='Reverse Limit Activated',sRcyText:='Reverse Limit Switch Is Activated. Reset The Error By Operate The Motor Backwards.')];
END_VAR
(**)
(*Local Output*)
VAR
	tyParamOut : tyMotionCANParamOut;
	sAxisErrTxt : STRING[80];
	bWidthPosDiff : BOOL;
	bJogOpen : BOOL;
	bJogClose : BOOL;
	bJogging : BOOL;
	bOpenSen : BOOL;
	bCloseSen : BOOL;
END_VAR
(**)
(*Local Input*)
VAR
	udiRstErr : UDINT := 0;
	bPrep : BOOL := TRUE;
	bEn : BOOL := TRUE;
	bDis : BOOL := FALSE;
	bOps : BOOL := FALSE;
	bManual : BOOL := FALSE;
	diWidthAtHmPos : DINT := 400;
	tyTuning : tyMotionCANTuning;
	diGoWidth : DINT := 150;
	diJogVelInUMPS : DINT := 10000;
	diMovePosInUM : DINT := 0;
	diMoveDistInUM : DINT := 0;
	diMoveVelInUMPS : DINT := 10000;
	diMoveAcc : DINT := 500;
	diMoveDec : DINT := 500;
	diMinAbsPosInUM : DINT := -3000;
	diMaxAbsPosInUM : DINT := 10000000;
	diMinWidthInUM : DINT := 70000;
	diMaxWidthInUM : DINT := 460000;
	diWidthOffsetInUM : DINT := 0;
	bInletSensor : BOOL;
	bOutletSensor : BOOL;
	bClearSensor : BOOL;
	bMiddleSensor : BOOL;
	bInterruptSensor : BOOL;
	bOpenInterruptSensor : BOOL;
	bCloseInterruptSensor : BOOL;
	bDir : BOOL;
	bDirBl : BOOL;
	bNoIndexPulse : BOOL;
	usiNode : USINT;
	sDevice : STRING[3];
	sProgNm : STRING[15] := 'AWOpen';
	diMoveBacklashDistInUM : DINT := 3000;
	diPitchInUM : DINT := 3000;
	tyParamInHm : tyMotionCANParamInHm;
	tyParamInConvert : tyMotionCANParamInConvert := (diPitchInUM:=3000);
	bNtSettingsLoadDone : BOOL := TRUE;
	eMotorType : eServoMotorType := DeltaAsdaA2;
END_VAR
(**)
(*Local*)
VAR
	bRstErr : BOOL;
	udiRstErrOld : UDINT;
	bInitDone : BOOL;
	bInitialDone : BOOL;
	bModuleOKChk : BOOL := TRUE;
	bModuleOK : BOOL;
	bModuleNotOK : BOOL := TRUE;
	bModuleNotOKLock : BOOL;
	bNotInterruptible : BOOL;
	bInterruptSensor1 : BOOL;
	bInterruptSensor2 : BOOL;
	diActualPosInUMOld : DINT;
	usiRstStep : USINT := 0;
	usiStep : USINT;
	usiCount : USINT;
	fbTm : TON := (PT:=T#2s);
	fbServoModuleNotOk : TON := (IN:=FALSE,PT:=T#2s);
	fbServoModuleOk : TON := (IN:=FALSE,PT:=T#5s);
	fbRstNodeTimer : TON := (PT:=T#3s);
	tyParamInMove : tyMotionCANParamInMove;
	tyParamInDriver : tyMotionCANDriverIn;
	tyParamOutDriver : tyMotionCANDriverOut := (siModOfOpt_6060:=6);
	fbStop : fbMotionCANStop;
	fbRstAxisErr : fbMotionCANRstAxisErr;
	fbJog : fbMotionCANJog;
	fbMovRel : fbMotionCANMovRel;
	fbMovAbs : fbMotionCANMovAbs;
	fbHoming : fbMotionCANHoming;
	fbPwrOff : fbMotionCANPwrOff;
	fbPwrOn : fbMotionCANPwrOn;
	fbFullHm : fbMotionCANFullHm;
	fbFullMovAbs : fbMotionCANFullMovAbs;
	fbFullMovAbsBl : fbMotionCANFullMovAbsBl;
	fbModuleOK : fbMotionCANModuleOK;
	fbSDOWrite : fbCANSDOWriteArrayParam;
	udiModuleNum : UDINT := 1;
END_VAR
```

### Trav.typ - Do Not Change!!!
```iecst
(*2018-12-27*)
(**)
(*Action*)

TYPE
	eTravAction :
		(
		TravActIdle,
		TravActGoAPos,
		TravActGoBPos,
		TravActGoCPos,
		TravActGoDPos,
		TravActGoEPos,
		TravActGoFPos,
		TravActGoGPos,
		TravActGoHPos,
		TravActFullHm,
		TravActPwrOn,
		TravActPwrOff,
		TravActHoming,
		TravActMovAbs,
		TravActMovRel,
		TravActJogFront,
		TravActJogRear,
		TravActJogStop,
		TravActRstAxisErr,
		TravActStop,
		TravActSDOWrite,
		TravActBGStartModOKChk,
		TravActBGStopModOKChk,
		TravActRstNode
		);
END_TYPE
```

### Trav.var - Change By Project
```iecst
(*2019-04-24*)
(**)
(*Action & State & Status*)
VAR
	p_TravStat : UDINT;
	p_TravStatus : UDINT;
	p_TravStatTxt : UDINT;
END_VAR
(**)
(*Alarm*)
VAR
	p_TravAlmData : UDINT;
	p_TravAlmData1 : UDINT;
	p_TravAlmData2 : UDINT;
	p_TravAlmData3 : UDINT;
END_VAR
(**)
(*Output*)
VAR
	p_TravParamOut : UDINT;
	p_TravPwrOn : UDINT;
	p_TravIsHomed : UDINT;
	p_TravPosDiff : UDINT;
	p_TravAxisErr : UDINT;
	p_TravAxisErrID : UDINT;
	p_TravAxisErrTxt : UDINT;
	p_TravFwdLmtSen : UDINT;
	p_TravRevLmtSen : UDINT;
	p_TravActualPos : UDINT;
	p_TravAPosDiff : UDINT;
	p_TravBPosDiff : UDINT;
	p_TravCPosDiff : UDINT;
	p_TravDPosDiff : UDINT;
	p_TravEPosDiff : UDINT;
	p_TravFPosDiff : UDINT;
	p_TravGPosDiff : UDINT;
	p_TravHPosDiff : UDINT;
	p_TravJogging : UDINT;
	p_TravFrontSen : UDINT;
	p_TravRearSen : UDINT;
END_VAR
```

### Program Logical/CANOpenServo/Trav/Trav (IEC, version 1.00.0) - 1.00.0 - NtMotion v5.00.0

#### Init.st - Change By Project
```iecst
(** 2019-04-24 **)
PROGRAM _INIT

	(* Always Change If Project Change *)

	//Pass Address To Global Address For External Use
	//Action, State & Status
	p_TravStat		:= ADR(eStat);
	p_TravStatus	:= ADR(eMainStatus);
	p_TravStatTxt	:= ADR(sStatTxt);

	//Alarm
	p_TravAlmData	:= ADR(tyAlmData);
	p_TravAlmData1	:= ADR(tyAlmData1);
	p_TravAlmData2	:= ADR(tyAlmData2);
	p_TravAlmData3	:= ADR(tyAlmData3);

	//Output
	p_TravParamOut		:= ADR(tyParamOut);
	p_TravPwrOn			:= ADR(tyParamOut.bPwrOn);
	p_TravIsHomed		:= ADR(tyParamOut.bIsHomed);
	p_TravPosDiff		:= ADR(tyParamOut.bPosDiff);
	p_TravAxisErr		:= ADR(tyParamOut.bAxisErr);
	p_TravAxisErrID		:= ADR(tyParamOut.udiAxisErrID);
	p_TravFwdLmtSen		:= ADR(tyParamOut.bFwdLmtSen);
	p_TravRevLmtSen		:= ADR(tyParamOut.bRevLmtSen);
	p_TravActualPos		:= ADR(tyParamOut.diActualPosInUM);
	p_TravAxisErrTxt	:= ADR(sAxisErrTxt);
	p_TravAPosDiff		:= ADR(bAPosDiff);
	p_TravBPosDiff		:= ADR(bBPosDiff);
	p_TravCPosDiff		:= ADR(bCPosDiff);
	p_TravDPosDiff		:= ADR(bDPosDiff);
	p_TravEPosDiff		:= ADR(bEPosDiff);
	p_TravFPosDiff		:= ADR(bFPosDiff);
	p_TravGPosDiff		:= ADR(bGPosDiff);
	p_TravHPosDiff		:= ADR(bHPosDiff);
	p_TravJogging		:= ADR(bJogging);
	p_TravFrontSen		:= ADR(bFrontSen);
	p_TravRearSen		:= ADR(bRearSen);

	(* Always Change If Project Change *)

END_PROGRAM
```

#### Act_InitGlobal.st - Change By Project
```iecst
(** 2019-04-09 **)
ACTION Act_InitGlobal:

	(* Always Change If Project Change *)

	//Pass Data To Link
	p_bLinkOpsRun ACCESS p_OpsRun;
	p_bLinkStartupRun ACCESS p_StartupRun;
	p_bSimu ACCESS p_UISimuMod;

	p_bLinkOpsTravLifULInDSPos ACCESS p_OpsTravLifULInDSPos;
	p_bLinkNtParamProjUsFixToFixRail ACCESS p_NtParamProjUsFixToFixRail;
	p_diLinkFixtoFixPosIn ACCESS p_McParamTravInletFixtoFixPos;
	p_diLinkMcParamTravPosB ACCESS p_McParamTravPosB;
	p_tyProdRcpCurrRcp ACCESS p_ProdRcpCurrRcp1;
	p_bLinkSafetyRelay ACCESS p_DISafetyRlySig;

	p_diLinkDPos ACCESS p_MagRcpCurrRcpMag1TravPos;
	p_diLinkEPos ACCESS p_MagRcpCurrRcpMag2TravPos;
	p_diLinkFPos ACCESS p_MagRcpCurrRcpMag3TravPos;

	p_bLinkTravGotoChkPt ACCESS p_OpsTravLifULTravGotoChkPt;
	p_diLinkTravGotoChkPtDist1 ACCESS p_McParamMag1WidthChkDetDist;
	p_diLinkTravGotoChkPtDist2 ACCESS p_McParamMag2WidthChkDetDist;
	p_diLinkTravGotoChkPtDist3 ACCESS p_McParamMag3WidthChkDetDist;

	//Pass Data To Internal Use
	p_udiRstErr ACCESS p_RstErrReset;
	p_bOps ACCESS p_OpsStatusRun;
	p_bManual ACCESS p_UIMnlMod;
	p_diAPos ACCESS p_McParamTravPosA;
//	p_diBPos ACCESS p_McParamTravPosB;
//	p_diDPos ACCESS p_MagRcpCurrRcpMag1TravPos;
//	p_diEPos ACCESS p_MagRcpCurrRcpMag2TravPos;
//	p_diFPos ACCESS p_MagRcpCurrRcpMag3TravPos;
	p_tyTuning ACCESS p_NtParamTravTuning;
	p_diJogVelInUMPS ACCESS p_UIMnlTravJogSpd;
	p_diMovePosInUM ACCESS p_UIMnlTravTargetPos;
	p_diMoveDistInUM ACCESS p_UIMnlTravStepSize;
	p_diMoveAcc ACCESS p_NtParamTravAcc;
	p_diMoveDec ACCESS p_NtParamTravDec;
	p_bDir ACCESS p_NtParamTravDir;
	p_usiNode ACCESS p_NtParamTravNode;
	p_sDevice ACCESS p_NtParamTravDevice;
	p_sProgNm ACCESS p_NtParamTravProgNm;
	p_tyParamInHm ACCESS p_NtParamTravParamInHm;
	p_tyParamInConvert ACCESS p_NtParamTravParamInConvert;
	p_bNtSettingsLoadDone ACCESS p_StartupNtSettingsLoadDone;
	p_eNtParamMotorType ACCESS p_NtParamTravMotorType;

	p_bInletShutterCloseRS ACCESS p_DIInShutterCloseRS;
	p_bOutletShutterCloseRS ACCESS p_DIOutShutterCloseRS;
	p_bOutletShutterCloseRS2 ACCESS p_DIOutShutterCloseRS2;
	p_bOutletShutterCloseRS3 ACCESS p_DIOutShutterCloseRS3;
	p_bProjInletShutPrep ACCESS p_NtParamProjInletShutPrep;
	p_bInShutterDis ACCESS p_McParamInShutterDis;
	p_bProjOutletShutPrep ACCESS p_NtParamProjOutletShutPrep;
	p_bPusherRetSen ACCESS p_DIPusherRetRS;
	p_bPusherExtSen ACCESS p_DIPusherExtRS;

	p_bDIConvLftSen ACCESS p_DIConvLftSen;
	p_bDIConvClrSen ACCESS p_DIConvClrSen;
	(* Always Change If Project Change *)

END_ACTION
```

#### InputRef_Link.var - Change By Project
```iecst
(*2019-04-09*)
(**)
(*External Data*)
VAR
	p_bLinkOpsRun : REFERENCE TO BOOL;
	p_bLinkStartupRun : REFERENCE TO BOOL;
	p_bSimu : REFERENCE TO BOOL;
	p_bLinkOpsTravLifULInDSPos : REFERENCE TO BOOL;
	p_bLinkNtParamProjUsFixToFixRail : REFERENCE TO BOOL;
	p_diLinkFixtoFixPosIn : REFERENCE TO DINT;
	p_diLinkMcParamTravPosB : REFERENCE TO DINT;
	p_tyProdRcpCurrRcp : REFERENCE TO tyProdRcpParam;
	p_bLinkSafetyRelay : REFERENCE TO BOOL;
	p_diLinkDPos : REFERENCE TO DINT;
	p_diLinkEPos : REFERENCE TO DINT;
	p_diLinkFPos : REFERENCE TO DINT;
	p_bLinkTravGotoChkPt : REFERENCE TO BOOL;
	p_diLinkTravGotoChkPtDist1 : REFERENCE TO DINT;
	p_diLinkTravGotoChkPtDist2 : REFERENCE TO DINT;
	p_diLinkTravGotoChkPtDist3 : REFERENCE TO DINT;
END_VAR
```

#### Act_LinkAction.st - Change By Project
```iecst
(** 2019-10-21 **)
ACTION Act_LinkAction:

	IF eStatus = Idle THEN
		IF bModuleNotOK THEN
			p_eAct ACCESS ADR(eAct);
		ELSE
			IF p_bLinkStartupRun = TRUE THEN
				p_eAct ACCESS p_StartupTravAct;
			ELSIF p_bLinkOpsRun = TRUE THEN
				p_eAct ACCESS p_OpsTravLifULTravAct;
			ELSIF p_bManual = TRUE OR p_bSimu THEN //
				p_eAct ACCESS p_UITravAct;
			ELSE
				p_eAct ACCESS ADR(eAct);
			END_IF
		END_IF
	END_IF

	IF EDGENEG(p_bManual) OR EDGENEG(p_bLinkOpsRun) OR EDGENEG(p_bLinkStartupRun) THEN
		tyParamOutDriver.uiCtrlword_6040	:= 0;
	END_IF

END_ACTION
```

#### Cyclic.st - Do Not Change!!!
```iecst
(** 2020-03-16 **)
PROGRAM _CYCLIC

	IF bInitDone = FALSE THEN
		bInitDone	:= TRUE;

		Act_InitLocal;
		Act_InitGlobal;

	ELSIF bInitialDone = FALSE THEN
		IF p_bNtSettingsLoadDone = TRUE THEN
			bInitialDone	:= TRUE;

			Act_Initial;
		END_IF

	ELSE

		Act_RstErr;
		Act_LinkAction;
		Act_Action;
		Act_LinkEn;

		IF (p_bPrep = TRUE) AND (p_bEn = TRUE) AND (p_bDis = FALSE) THEN
			Act_Link;
			Act_Background;
			Act_Main;
		ELSE
			Act_Main_Disable;

			IF eStat <> TravActIdle THEN
				eStatus	:= Done;
			ELSE
				eStatus	:= Idle;
			END_IF
		END_IF

		Act_CombineErr;
		Act_Alarm;
		Act_Alarm1;
		Act_Alarm2;
		Act_Alarm3;

	END_IF

END_PROGRAM
```

#### Act_Link.st - Change By Project
```iecst
(** 2019-03-29 **)
ACTION Act_Link:

	IF p_bManual = TRUE THEN
		p_diMoveVelInUMPS ACCESS p_UIMnlTravNomSpd;
	ELSE
		p_diMoveVelInUMPS ACCESS p_NtParamTravAutoSpd;
	END_IF

	IF p_bProjInletShutPrep = TRUE AND p_bInShutterDis = FALSE AND p_bLinkOpsTravLifULInDSPos = FALSE AND (p_bOps OR p_bManual) THEN

		IF (p_bInletShutterCloseRS = FALSE AND NOT p_bOps) OR p_bPusherRetSen = FALSE OR p_bPusherExtSen
			THEN
			p_bInterruptSensor1 := TRUE;
		ELSE
			p_bInterruptSensor1 := FALSE;
		END_IF
	ELSE
		p_bInterruptSensor1 := FALSE;
	END_IF

	IF p_bProjOutletShutPrep = TRUE AND p_bLinkOpsTravLifULInDSPos = FALSE THEN
		IF ((p_bOutletShutterCloseRS = FALSE OR p_bOutletShutterCloseRS2 = FALSE OR p_bOutletShutterCloseRS3 = FALSE) AND NOT p_bOps) OR p_bPusherRetSen = FALSE OR p_bPusherExtSen
			THEN
			p_bInterruptSensor2 := TRUE;
		ELSE
			p_bInterruptSensor2 := FALSE;
		END_IF
	ELSE
		p_bInterruptSensor2 := FALSE;
	END_IF

//	IF p_bDIConvLftSen OR p_bDIConvClrSen THEN
//		p_bInterruptSensor3 := TRUE;
//	ELSE
//		p_bInterruptSensor3 := FALSE;
//	END_IF

	//Add

	IF NOT p_bOps THEN
		p_bInterruptSensor1	:= FALSE;
		p_bInterruptSensor2 := FALSE;

	END_IF

	IF p_bLinkNtParamProjUsFixToFixRail THEN
		p_diBPos := p_diAPos + p_diLinkFixtoFixPosIn - p_tyProdRcpCurrRcp.diWidthInUM;
	ELSE
		p_diBPos := p_diLinkMcParamTravPosB;
	END_IF

	IF p_bLinkTravGotoChkPt THEN // To Check the Magazine Width - Offset of Traverser
		p_diDPos := p_diLinkDPos + p_diLinkTravGotoChkPtDist1;
		p_diEPos := p_diLinkEPos + p_diLinkTravGotoChkPtDist2;
		p_diFPos := p_diLinkFPos + p_diLinkTravGotoChkPtDist3;
	ELSE
		p_diDPos := p_diLinkDPos;
		p_diEPos := p_diLinkEPos;
		p_diFPos := p_diLinkFPos;
	END_IF

//	p_bInterruptSensor3 := p_bLinkSafetyRelay = FALSE;

END_ACTION
```

#### Act_InitLocal.st - Change By Project
```iecst
(** 2020-03-16 **)
ACTION Act_InitLocal:

	//Input Reference Link To Local Variable
	p_eAct ACCESS ADR(eAct);
	p_udiRstErr ACCESS ADR(udiRstErr);
	p_bPrep ACCESS ADR(bPrep);
	p_bEn ACCESS ADR(bEn);
	p_bDis ACCESS ADR(bDis);
	p_bOps ACCESS ADR(bOps);
	p_bManual ACCESS ADR(bManual);
	p_diAPos ACCESS ADR(diAPos);
	p_diBPos ACCESS ADR(diBPos);
	p_diCPos ACCESS ADR(diCPos);
	p_diDPos ACCESS ADR(diDPos);
	p_diEPos ACCESS ADR(diEPos);
	p_diFPos ACCESS ADR(diFPos);
	p_diGPos ACCESS ADR(diGPos);
	p_diHPos ACCESS ADR(diHPos);
	p_tyTuning ACCESS ADR(tyTuning);
	p_diJogVelInUMPS ACCESS ADR(diJogVelInUMPS);
	p_diMovePosInUM ACCESS ADR(diMovePosInUM);
	p_diMoveDistInUM ACCESS ADR(diMoveDistInUM);
	p_diMoveVelInUMPS ACCESS ADR(diMoveVelInUMPS);
	p_diMoveAcc ACCESS ADR(diMoveAcc);
	p_diMoveDec ACCESS ADR(diMoveDec);
	p_diMinAbsPosInUM ACCESS ADR(diMinAbsPosInUM);
	p_diMaxAbsPosInUM ACCESS ADR(diMaxAbsPosInUM);
	p_bInterruptSensor1 ACCESS ADR(bInterruptSensor1);
	p_bInterruptSensor2 ACCESS ADR(bInterruptSensor2);
	p_bInterruptSensor3 ACCESS ADR(bInterruptSensor3);
	p_bInterruptSensor4 ACCESS ADR(bInterruptSensor4);
	p_bInterruptSensor5 ACCESS ADR(bInterruptSensor5);
	p_bDir ACCESS ADR(bDir);
	p_bNoIndexPulse ACCESS ADR(bNoIndexPulse);
	p_usiNode ACCESS ADR(usiNode);
	p_sDevice ACCESS ADR(sDevice);
	p_sProgNm ACCESS ADR(sProgNm);
	p_tyParamInHm ACCESS ADR(tyParamInHm);
	p_tyParamInConvert ACCESS ADR(tyParamInConvert);
	p_bNtSettingsLoadDone ACCESS ADR(bNtSettingsLoadDone);

	p_bInletShutterCloseRS ACCESS ADR(bInletShutterCloseRS);
	p_bOutletShutterCloseRS ACCESS ADR(bOutletShutterCloseRS);

	p_bProjInletShutPrep ACCESS ADR(bProjInletShutPrep);
	p_bInShutterDis ACCESS ADR(bInShutterDis);
	p_bProjOutletShutPrep ACCESS ADR(bProjOutletShutPrep);

END_ACTION
```

#### Act_Initial.st - Do Not Change!!!
```iecst
(** 2020-03-16 **)
ACTION Act_Initial:

	//Initial
	sStatTxt	:= a_sStatText[eStat];

	tyParamInMove.diAcc	:= p_diMoveAcc;
	tyParamInMove.diDec	:= p_diMoveDec;

	fbModuleOK.sDevice	:= p_sDevice;
	fbModuleOK.usiNode	:= p_usiNode;
	fbModuleOK.tDlyTm	:= T#5s;
	fbModuleOK(bEn := FALSE);

	fbSDOWrite.sDevice	:= p_sDevice;
	fbSDOWrite.usiNode	:= p_usiNode;
	fbSDOWrite.eMotorType	:= p_eNtParamMotorType;
	fbSDOWrite(bEn := FALSE);

	fbFullMovAbs.p_tyParamOutDriver		:= ADR(tyParamOutDriver);
	fbFullMovAbs.tyParamInMove.diAcc	:= p_diMoveAcc;
	fbFullMovAbs.tyParamInMove.diDec	:= p_diMoveDec;
	fbFullMovAbs.tyParamInConvert		:= p_tyParamInConvert;
	fbFullMovAbs.bDir					:= p_bDir;
	fbFullMovAbs.bNoIndexPulse			:= p_bNoIndexPulse;
	fbFullMovAbs.eMotorType				:= p_eNtParamMotorType;
	fbFullMovAbs(bEn := FALSE);

	fbFullHm.p_tyParamOutDriver	:= ADR(tyParamOutDriver);
	fbFullHm.bDir				:= p_bDir;
	fbFullHm.bNoIndexPulse		:= p_bNoIndexPulse;
	fbFullHm.eMotorType			:= p_eNtParamMotorType;
	fbFullHm(bEn := FALSE);

	fbPwrOn.p_tyParamOutDriver	:= ADR(tyParamOutDriver);
	fbPwrOn.eMotorType			:= p_eNtParamMotorType;
	fbPwrOn(bEn := FALSE);

	fbPwrOff.p_tyParamOutDriver	:= ADR(tyParamOutDriver);
	fbPwrOff.eMotorType			:= p_eNtParamMotorType;
	fbPwrOff(bEn := FALSE);

	fbHoming.p_tyParamOutDriver	:= ADR(tyParamOutDriver);
	fbHoming.bDir				:= p_bDir;
	fbHoming.bNoIndexPulse		:= p_bNoIndexPulse;
	fbHoming.eMotorType			:= p_eNtParamMotorType;
	fbHoming(bEn := FALSE);

	fbMovAbs.p_tyParamOutDriver		:= ADR(tyParamOutDriver);
	fbMovAbs.tyParamInMove.diAcc	:= p_diMoveAcc;
	fbMovAbs.tyParamInMove.diDec	:= p_diMoveDec;
	fbMovAbs.tyParamInConvert		:= p_tyParamInConvert;
	fbMovAbs.bDir					:= p_bDir;
	fbMovAbs.eMotorType				:= p_eNtParamMotorType;
	fbMovAbs(bEn := FALSE);

	fbMovRel.p_tyParamOutDriver		:= ADR(tyParamOutDriver);
	fbMovRel.tyParamInMove.diAcc	:= p_diMoveAcc;
	fbMovRel.tyParamInMove.diDec	:= p_diMoveDec;
	fbMovRel.tyParamInConvert		:= p_tyParamInConvert;
	fbMovRel.bDir					:= p_bDir;
	fbMovRel.eMotorType				:= p_eNtParamMotorType;
	fbMovRel(bEn := FALSE);

	fbJog.p_tyParamOutDriver	:= ADR(tyParamOutDriver);
	fbJog.tyParamInConvert		:= p_tyParamInConvert;
	fbJog.eMotorType			:= p_eNtParamMotorType;
	fbJog(bEn := FALSE);

	fbRstAxisErr.p_tyParamOutDriver	:= ADR(tyParamOutDriver);
	fbRstAxisErr(bEn := FALSE);

	fbStop.p_tyParamOutDriver	:= ADR(tyParamOutDriver);
	fbStop(bEn := FALSE);

	bModuleNotOK	:= TRUE;
END_ACTION
```

#### Act_Action.st - Do Not Change!!!
```iecst
(** 2020-03-16 **)
ACTION Act_Action:

	//Reset Error
	IF (eStatus = Error) AND bRstErr THEN
		p_eAct	:= TravActIdle;
		eStat	:= TravActIdle;

		fMotionCANRstCtrlWord(ADR(tyParamOutDriver));
	END_IF

	//Reset Done
	IF eStatus = Done AND p_eAct = TravActIdle THEN
		eStat	:= TravActIdle;
	END_IF

	//Set p_eAct
	IF (eStatus = Idle AND eStatus1 = Idle AND eStatus2 = Idle AND eStatus3 = Idle) OR p_eAct = TravActIdle OR p_eAct = TravActStop OR p_eAct = TravActJogStop THEN
		eStat	:= p_eAct;
	END_IF

END_ACTION
```
